// TIA Portal V17 program export: 1 tag tables, 0 data types, 0 data blocks, 3 code blocks (in call order from the OBs), 1 instance data blocks

VAR_GLOBAL   // PLC tag table "Default tag table"
   Sw1 AT %I0.0 : Bool;
   Sw2 AT %I0.1 : Bool;
   Output1 AT %Q0.0 : Bool;
   Output2 AT %Q0.1 : Bool;
END_VAR

ORGANIZATION_BLOCK "Main"   // OB1, LAD, ProgramCycle
TITLE = "Main Program Sweep (Cycle)"
{ S7_Optimized_Access := 'TRUE' }
VERSION : 0.1
// stored: AutoNumber true, IsIECCheckEnabled false, SetENOAutomatically false
   VAR_INPUT
      Initial_Call : Bool;   // Initial call of this OB
      Remanence : Bool;   // =True, if remanent data are available
   END_VAR
BEGIN

REGION Network 1
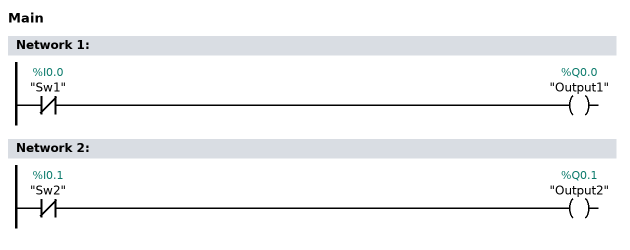
   RUNG wire#powerrail
      I_Contact( "Sw1" )
      Coil( "Output1" )
   END_RUNG
   // the same network as SCL:
   "Output1" := NOT "Sw1";
END_REGION

REGION Network 2
   RUNG wire#powerrail
      I_Contact( "Sw2" )
      Coil( "Output2" )
   END_RUNG
   // the same network as SCL:
   "Output2" := NOT "Sw2";
END_REGION
END_ORGANIZATION_BLOCK

FUNCTION "Block_1" : Void   // FC1, LAD
{ S7_Optimized_Access := 'TRUE' }
VERSION : 0.1
// stored: AutoNumber true, IsIECCheckEnabled false, SetENOAutomatically false, UDAEnableTagReadback false
BEGIN
END_FUNCTION

FUNCTION_BLOCK "Main_Safety_RTG1"   // FB1, F_FBD
{ S7_Optimized_Access := 'TRUE' }
VERSION : 0.1
// stored: AutoNumber false, IsIECCheckEnabled false, UDAEnableTagReadback false
BEGIN
END_FUNCTION_BLOCK

DATA_BLOCK "Main_Safety_RTG1_DB"   // DB1, F_DB
NAME : FUSI
VERSION : 0.1
// stored: AutoNumber true, InstanceOfName Main_Safety_RTG1, InstanceOfType FB
"Main_Safety_RTG1"
BEGIN
END_DATA_BLOCK
